{attribute 'GeneratedUsingTerminal: KL2022'}
{attribute addProperty BoxType "KL2022"}
{attribute addProperty Id "Channel_1AT %Q*Channel_460B8C400Channel_2AT %Q*Channel_460B8C400"}
{attribute addProperty CRC "3701954066"}
{attribute addProperty Size "0"}
TYPE KL2022_DCA75612 :
STRUCT
	{attribute addProperty Name "Channel_1"}
	Channel_1 : Channel_460B8C40;
	{attribute addProperty Name "Channel_2"}
	Channel_2 : Channel_460B8C40;
END_STRUCT
END_TYPE
